// TIA Portal V19 export
DATA_BLOCK "fbPnPnLeftCouplerDiag_DB"   // DB13
// stored: InstanceOfName fbGetDiagPnPnCouplerDiag, InstanceOfType FB
"fbGetDiagPnPnCouplerDiag"
   // VAR_INPUT
   //    LADDR : HW_ANY;
   //    DebounceTimer : Time;
   // END_VAR
   // VAR_OUTPUT
   //    OwnState : UInt;
   //    SubordinateState : UInt;
   //    DeviceStatusOk : Bool;
   // END_VAR
   // VAR
   //    Diag : DIS;
   //    Sub { S7_SetPoint := 'True'} : DNN;
   //    RetValueDiag : Int;
   //    CntDiagDiag : UInt;
   //    RetValueSub : Int;
   //    CntDiagSub : UInt;
   //    BadStateDebounceTimer : IEC_TIMER;
   // END_VAR
BEGIN
END_DATA_BLOCK
